{attribute 'qualified_only'}
{attribute 'strict'}
TYPE EMaterialPresence :
(
	Unknown := 0,
	Present,
	NotPresent
);
END_TYPE

(* stored: Version 1.1.0.1, ProductVersion 3.1.4024.12
   DUT EMaterialPresence: Id {87b1df0d-b1cf-4e12-9e9f-f5b922f7a811} *)
